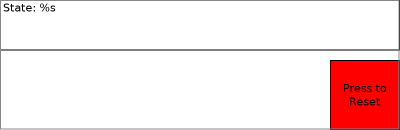
VISUALIZATION Vi_Safety  // 400x130
VAR_IN_OUT
	hmi		: Safety_Hmi;
END_VAR
    Rectangle (0,0 400x50), "State: %s", text variable: hmi.sStatusText
        p55702900: hmi.nStatusTextColor
    Rectangle (330,60 70x70), "Press to Reset", invisible if: NOT hmi.bResetButtonVis
        toggle hmi.bResetButton
END_VISUALIZATION

(* stored: Version 1.1.0.1
   Visu Vi_Safety: Id {d87a8060-5a5a-4c7e-a4fd-f1e76dffc94f} *)
